// Mitsubishi GX Works2 project: TIMEREX1   PLC: Q03UDV

PROGRAM MAIN
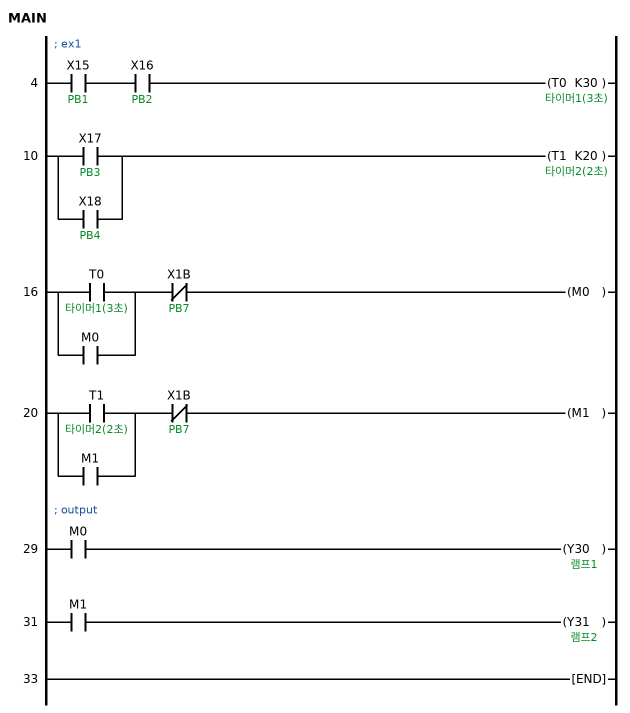
; ex1
4     LD      X15  ; PB1
      AND     X16  ; PB2
      OUT     T0 K30  ; 타이머1(3초)
10    LD      X17  ; PB3
      OR      X18  ; PB4
      OUT     T1 K20  ; 타이머2(2초)
16    LD      T0  ; 타이머1(3초)
      OR      M0
      ANI     X1B  ; PB7
      OUT     M0
20    LD      T1  ; 타이머2(2초)
      OR      M1
      ANI     X1B  ; PB7
      OUT     M1
; output
29    LD      M0
      OUT     Y30  ; 램프1
31    LD      M1
      OUT     Y31  ; 램프2
33    END
END_PROGRAM

// device comments not shown above
Y38  ; 실린더 전진
Y39  ; 실린더 후진
